// TwinCAT 3 PLC project TimeDelta
// ProgramVersion: 3.1.4023.0
// libraries:
//   Tc2_Standard, * (Beckhoff Automation GmbH)
//   Tc2_System, * (Beckhoff Automation GmbH)
//   Tc2_Utilities, * (Beckhoff Automation GmbH)
//   Tc3_Module, * (Beckhoff Automation GmbH)
// project tree:
//   DUTs/ ST_TimeStruct.TcDUT
//   / PlcTask.TcTTO
//   POUs/ FB_TimeDelta.TcPOU, F_GetSystemTime.TcPOU, MAIN.TcPOU
// real-time tasks:
//   TASK PlcTask: cycle T#10ms, priority 20, ADS port 350

CONFIGURATION TimeDelta
    RESOURCE PLC ON TwinCAT3
        TASK PlcTask(INTERVAL := T#10ms, PRIORITY := 20);
        PROGRAM MAIN WITH PlcTask : MAIN;
    END_RESOURCE
END_CONFIGURATION

// ---- DUTs/ST_TimeStruct.TcDUT
TYPE ST_TimeStruct :
STRUCT
	wYear : WORD;
    wMonth : WORD;
    wDayOfWeek : WORD;
    wDay : WORD;
    wHour : WORD;
    wMinute : WORD;
    wSecond : WORD;
    wMilliseconds : WORD;
END_STRUCT
END_TYPE

// ---- POUs/MAIN.TcPOU
PROGRAM MAIN
VAR
	fbTimeDelta : FB_TimeDelta;
	bStartButton : BOOL;
	bStopButton : BOOL;
	DisplayDeltaTime : ST_TimeStruct;
	bStartButtonPressed : BOOL := FALSE; // Latch for Start button
    bStopButtonPressed : BOOL := FALSE;  // Latch for Stop button
END_VAR

fbTimeDelta();

// Logic for Start Button
IF bStartButton AND NOT bStartButtonPressed THEN
    fbTimeDelta.Start(); // Record the start time
    bStartButtonPressed := FALSE; // Latch the start button
END_IF

// Reset the latch if the button is released
IF NOT bStartButton THEN
    bStartButtonPressed := FALSE;
END_IF

// Logic for Stop Button
IF bStopButton AND NOT bStopButtonPressed THEN
    fbTimeDelta.Stop(); // Record the stop time
    bStopButtonPressed := TRUE; // Latch the stop button
    
    // Calculate and display the delta time
    DisplayDeltaTime := fbTimeDelta.GetDelta();
END_IF

// Reset the latch if the button is released
IF NOT bStopButton THEN
    bStopButtonPressed := FALSE;
END_IF

END_PROGRAM

// ---- POUs/FB_TimeDelta.TcPOU
FUNCTION_BLOCK FB_TimeDelta
VAR
	StartTime : ST_TimeStruct;
    StopTime : ST_TimeStruct;
    CurrentTime : ST_TimeStruct; // Assuming this to be cyclically updated to the current PLC time
	fbGetSystemTime : GETSYSTEMTIME;
    timeAsFileTime : T_FILETIME;
    timeAsDT : DATE_AND_TIME;
END_VAR

F_GetSystemTime(F_GetSystemTime => CurrentTime);
GetDelta();

METHOD GetDelta : ST_TimeStruct
VAR
	DeltaTime : ST_TimeStruct;
END_VAR
// Calculate the delta TIME here AND assign it TO DeltaTime
	DeltaTime.wYear := StopTime.wYear - StartTime.wYear;
    DeltaTime.wMonth := StopTime.wMonth - StartTime.wMonth;
    DeltaTime.wDay := StopTime.wDay - StartTime.wDay;
    DeltaTime.wHour := StopTime.wHour - StartTime.wHour;
    DeltaTime.wMinute := StopTime.wMinute - StartTime.wMinute;
    DeltaTime.wSecond := StopTime.wSecond - StartTime.wSecond;
    DeltaTime.wMilliseconds := StopTime.wMilliseconds - StartTime.wMilliseconds;
	
// Adjust for negative values
    IF DeltaTime.wMilliseconds < 0 THEN
        DeltaTime.wMilliseconds := DeltaTime.wMilliseconds + 1000;
        DeltaTime.wSecond := DeltaTime.wSecond - 1;
    END_IF;
    IF DeltaTime.wSecond < 0 THEN
        DeltaTime.wSecond := DeltaTime.wSecond + 60;
        DeltaTime.wMinute := DeltaTime.wMinute - 1;
    END_IF;
    IF DeltaTime.wMinute < 0 THEN
        DeltaTime.wMinute := DeltaTime.wMinute + 60;
        DeltaTime.wHour := DeltaTime.wHour - 1;
    END_IF;
    IF DeltaTime.wHour < 0 THEN
        DeltaTime.wHour := DeltaTime.wHour + 24;
        DeltaTime.wDay := DeltaTime.wDay - 1;
    END_IF;
    // Handle month and year adjustments as needed

    GetDelta := DeltaTime;
END_METHOD

METHOD Start : ST_TimeStruct
VAR
END_VAR
// Assume CurrentTime is updated externally and cyclically with the current PLC time
F_GetSystemTime(F_GetSystemTime => StartTime);
END_METHOD

METHOD Stop : ST_TimeStruct
VAR
END_VAR
// Assume CurrentTime is updated externally and cyclically with the current PLC time
F_GetSystemTime(F_GetSystemTime => StopTime);
END_METHOD

END_FUNCTION_BLOCK

// ---- POUs/F_GetSystemTime.TcPOU
FUNCTION F_GetSystemTime : ST_TimeStruct
VAR
	fbGetSystemTime : GETSYSTEMTIME; 
    fileTime        : T_FILETIME;
    sDT: STRING(30);
END_VAR

fbGetSystemTime(timeLoDW => fileTime.dwLowDateTime, timeHiDW => fileTime.dwHighDateTime);
sDT := SYSTEMTIME_TO_STRING(FILETIME_TO_SYSTEMTIME(fileTime));

F_GetSystemTime.wYear := STRING_TO_WORD(LEFT(sDt, 4));
F_GetSystemTime.wMonth := STRING_TO_WORD(MID(sDt, 2, 6));
F_GetSystemTime.wDay := STRING_TO_WORD(MID(sDt, 2, 9));
F_GetSystemTime.wHour := STRING_TO_WORD(MID(sDt, 2, 12));
F_GetSystemTime.wMinute := STRING_TO_WORD(MID(sDt, 2, 15));
F_GetSystemTime.wSecond := STRING_TO_WORD(MID(sDt, 2, 18));
F_GetSystemTime.wMilliseconds := STRING_TO_WORD(RIGHT(sDt, 3));

END_FUNCTION
